{attribute 'Tc2GvlVarNames'}
VAR_CONFIG
END_VAR

(* stored: Version 1.1.0.1, ProductVersion 3.1.4024.15
   GVL Variable_Configuration: Id {ac798428-bda4-44f8-b8ab-2f00e23503b6} *)
